(* CoDeSys 2.3 export: SDO SVR CAN Preprocessor IFM NT.ST *)

(* POU SDO Server/FB_SDOSVR_CAN_NT, ST *)
FUNCTION_BLOCK FB_SDOSVR_CAN_NT (* SDO Server Interface for IFM NT hardware *)
VAR_INPUT
	CHANNEL : BYTE; (* CAN channel as required by CAN RX/TX *)
	NodeID_Init : USINT; (* Node ID to Initialize *)
	Enum_RX : POINTER TO FB_SDOSVR_CAN_NT_ENUM_RX; (* optional enumeration request receiver block *)
	Enum_RX_Flag : BOOL; (* Enumeration request to receive and process? *)
	SDOSVR_PROC : FB_SDOSVR_PROC; (* instance of an SDO server processor *)
END_VAR
VAR_OUTPUT
	INIT : BOOL := TRUE; (* block needs initialized? *)
	NodeID_Set : USINT; (* Node ID currently set *)
	TX_BUFFER_FULL : BOOL; (* TX_BUFFER was full, TX couldn't be made, need to wait for more room *)
	RX_BUFFER_EMPTY : BOOL; (* RX_BUFFER was empty, no need for further processing *)
END_VAR
VAR
	RX_CAN : CAN_RX_ENH_FIFO := ( ENABLE:=TRUE, ID_MASK:=16#7FF ); (* IFM NT CAN receive block *)
	TX_CAN : CAN_TX_ENH := ( ENABLE:=TRUE ); (* IFM NT CAN transmit block *)
	(* V1-1 removed Chk_Timers, revised scheme doesn't require the flag *)
END_VAR
IF NOT INIT THEN
	REPEAT
		(* check if action left with pending transmit *)
		IF SDOSVR_PROC.CANSDO_TX THEN
			TX_CAN( DATA:=SDOSVR_PROC.CANSDO_DATA, DATALENGTHCODE:=SDOSVR_PROC.CANSDO_DLC );
			TX_BUFFER_FULL := TX_CAN.RESULT = 250; (* track if TX FIFO is full *)
			IF NOT TX_BUFFER_FULL THEN
				SDOSVR_PROC.CLEAR_TX_REQ; (* clear TX flag and clean up previous request results or pending actions *)
			ELSIF Enum_RX_Flag THEN (* added 2018-06-19 CMM, moved to TX section 2018-11-02 CMM *)
				(* Enumeration request was pending, but with no way to respond to it, we must abandon it *)
				Enum_RX_Flag := FALSE;
			END_IF
		ELSE
			SDOSVR_PROC.CleanUp; (* clean up any previous request results and pending actions, sending INV_OBJ if required (generating another transmit) *)
		END_IF

		(* if a pending transmit is still pending, we cannot process any received messages, as they may cause transmission requests *)
		IF SEL( SDOSVR_PROC.CANSDO_TX, SDOSVR_PROC.Request_RESULT <= 1, FALSE ) THEN
			(* all seems to be good, check RX, and if any, attempt to process *)
			RX_CAN;
			RX_BUFFER_EMPTY := NOT RX_CAN.MORE_DATA_AVAILABLE;
			IF RX_CAN.RESULT = 1 OR RX_CAN.RESULT = 250 THEN
				SDOSVR_PROC( CANSDO_DATA:=RX_CAN.DATA, CANSDO_DLC:=RX_CAN.DATALENGTHCOUNT );
			ELSIF Enum_RX_Flag THEN
				IF Enum_RX <> 0 THEN
					(* process enumeration request *)
					SDOSVR_PROC( CANSDO_DATA:=Enum_RX^.RX_CAN.DATA, CANSDO_DLC:=Enum_RX^.RX_CAN.DATALENGTHCOUNT, CANSDO_IsEnum:=TRUE );
				END_IF
				Enum_RX_Flag := FALSE;
			END_IF
			IF SEL( SDOSVR_PROC.Request_RESULT = 1, FALSE, SEL( SDOSVR_PROC.CANSDO_TX, RX_BUFFER_EMPTY, FALSE ) ) THEN
				(* SDO service has active transfers, but is presently idle, check transfer timers *)
				SDOSVR_PROC.ChkTimers; (* need to process timers, aborting transfers if timers have expired *)
			END_IF
		END_IF

	(* as long as TX FIFO isn't full and SDO processor is not pending a dispatch, if SDO processor still pending a TX OR CAN buffer has more data, repeat loop in attempt to clear it *)
	UNTIL SEL( TX_BUFFER_FULL, SEL( SDOSVR_PROC.Request_RESULT > 1, NOT (SDOSVR_PROC.CANSDO_TX OR Enum_RX_Flag) AND RX_BUFFER_EMPTY, TRUE ), TRUE )
	END_REPEAT
ELSE
	TX_BUFFER_FULL := TRUE; (* we are not initialized, so the TX buffer is considered full *)
END_IF
END_FUNCTION_BLOCK
ACTION InitSvr:
(* Initialize server, should cancel any pending operations, though not neccessary *)
RX_CAN.CHANNEL := TX_CAN.CHANNEL := CHANNEL; (* set which NT channel to operate on *)
NodeID_Set := MIN( NodeID_Init, 127 ); (* restrict range of node ID's *)
RX_CAN.ID := 16#600 + NodeID_Set; (* specify desired SDO request ID *)
TX_CAN.ID := 16#580 + NodeID_Set; (* specify desired SDO response ID *)
Enum_RX_Flag := SDOSVR_PROC.CANSDO_IsEnum := FALSE; (* clarifying startup condition *)
INIT := FALSE; (* done initialized *)
END_ACTION
